TYPE DUT_Example :
STRUCT
END_STRUCT
END_TYPE

(* stored: Version 1.1.0.1, ProductVersion 3.1.4022.18
   DUT DUT_Example: Id {a09844c4-1872-4a30-a6e9-6cce686fe5e1} *)
